FUNCTION_BLOCK FB_Picker_2 EXTENDS FB_Picker
VAR_INPUT
END_VAR
VAR_OUTPUT
END_VAR
VAR
END_VAR

SUPER^();

METHOD M_MoveToPickPos : BOOL
VAR_INPUT
	Buffer_1_InUse : BOOL;
	Buffer_Pos : INT;
END_VAR
//If Mover1 then PickFromCassette; if Mover2  PickFromBuffer

//State := E_MoverTransitionState.Picking;


Sim_Time(IN := TRUE, PT := T#1S);

IF Sim_Time.Q THEN       //We assume in 1 seconds we go to Pick position; CassettePos for Mover1, BufferPos for Mover2
	Sim_Time(IN := FALSE);
	State := E_PickerFixedState.InPickedPos;
END_IF
END_METHOD

METHOD M_MoveToPlacePos : BOOL
//If Mover1 then PlaceToCarrier; if Mover2  PlaceToBuffer
//State := E_MoverTransitionState.Placing;


Sim_Time(IN := TRUE, PT := T#1S);

IF Sim_Time.Q THEN   //We assume in 1 seconds we go to Pick position; BufferPos for Mover1, CarrierPos for Mover2
	Sim_Time(IN := FALSE);
	State := E_PickerFixedState.InPlacedPos;
END_IF
END_METHOD

END_FUNCTION_BLOCK

(* stored: Version 1.1.0.1, ProductVersion 3.1.4024.12
   POU FB_Picker_2: Id {ae141df9-b1af-4fb5-8cce-8c6c54822038}, SpecialFunc None
   Folder Public: Id {af285bc4-b00c-4a4e-9e52-036d5d6a95cd}
   Method M_MoveToPickPos: Id {e258428f-1e1d-4ad3-a463-236cc2a4631c}
   Method M_MoveToPlacePos: Id {0dc6fcdf-22f9-4ad6-8f31-34f2d76363ff} *)
